FUNCTION_BLOCK FB_Beckhoff_EL5152_Test EXTENDS TcUnit.FB_TestSuite
VAR
	fbDevice : FB_Beckhoff_EL5152;
	nExpected : UINT;
	nResult : UINT;
END_VAR

TEST('nCounter1');
nExpected := 111;
fbDevice.nValue1 := nExpected;
fbDevice();
nResult := fbDevice.Counter1;
AssertEquals(Expected := nExpected,
             Actual := nResult,
             Message := 'nCounter1 value is not correct');	
TEST_FINISHED();

TEST('nCounter2');
nExpected := 112;
fbDevice.nValue2 := nExpected;
fbDevice();
nResult := fbDevice.Counter2;
AssertEquals(Expected := nExpected,
             Actual := nResult,
             Message := 'nCounter2 value is not correct');	
TEST_FINISHED();


TEST('nStatus1');
nExpected := 4;
fbDevice.Control1 := nExpected;
fbDevice();
nResult := fbDevice.Status1;
AssertEquals(Expected := nExpected,
             Actual := nResult,
             Message := 'nStatus1 value is not correct');	
TEST_FINISHED();

TEST('nStatus2');
nExpected := 4;
fbDevice.Control2 := nExpected;
fbDevice();
nResult := fbDevice.Status2;
AssertEquals(Expected := nExpected,
             Actual := nResult,
             Message := 'nStatus2 value is not correct');	
TEST_FINISHED();

END_FUNCTION_BLOCK

(* stored: Version 1.1.0.1, ProductVersion 3.1.4024.12
   POU FB_Beckhoff_EL5152_Test: Id {41eadc21-428a-091f-0416-55b3c1826864}, SpecialFunc None *)
